Staubli VAL3: check_cylinder.pgx

public program check_cylinder(tool x_tTool, bool& x_bCheck[])
  local point l_pPoint
  local point l_pNewOrigin
begin
  //
  // CHECK IF THE TOOL IS INSIDE
  //
  x_bCheck=false
  //
  if bCreate_cylind
    l_pPoint=here(x_tTool,fCube)
    // check if inside
    if l_pPoint.trsf.z>=-0.1 and l_pPoint.trsf.z<=nDistanceZ_cyl
      // inside the cylinder
      l_pNewOrigin=compose(pOrigin_cylind,world,{0,0,l_pPoint.trsf.z,0,0,0})
      if distance(l_pNewOrigin,l_pPoint)<=nRadius_cyl
        // is inside
        x_bCheck=true
      endIf
    endIf
  endIf
end
